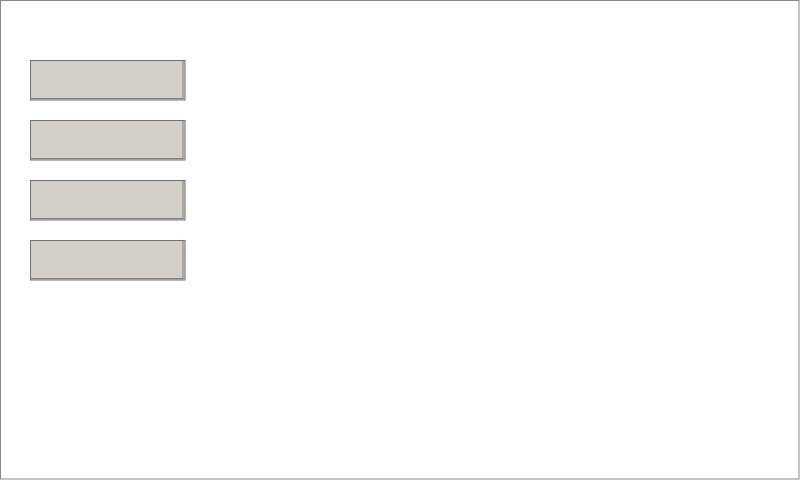
VISUALIZATION Main  // 800x480, background image ImagePool.homeScreen
    Button (30,60 155x40), image: Buttons.manualButton
        OnMouseClick: change screen: manualMode
    Button (30,120 155x40), image: Buttons.automaticButton
        OnMouseDown: change screen: autoMode
    Button (30,180 155x40), image: Buttons.controlButton
        OnMouseClick: change screen: allControls
        OnMouseClick: execute { MAIN.allControls:=TRUE; }
    Button (30,240 155x40), image: Buttons.aboutButton
        OnMouseClick: change screen: about
END_VISUALIZATION

(* stored: Version 1.1.0.1, ProductVersion 3.1.4018.2
   Visu Main: Id {eb4955ea-4d9d-4dcf-939b-6a17521bc80f} *)
